Yaskawa INFORM job: OK_R2_O24A(90,180)OKKR.JBI

/JOB
//NAME OK_R2_O24A(90,180)OKKR
///FOLDERNAME X4
//POS
///NPOS 233,233,233,10,0,0
///TOOL 0
///POSTYPE PULSE
///PULSE
C00000=127652,-120361,-107124,-61599,94745,-41314
C00001=123475,-119595,-103586,-61416,91214,-41301
C00002=121798,-119103,-102107,-61373,89825,-41321
C00003=122733,-118069,-99629,-61351,89920,-40763
C00004=120759,-117967,-99269,-61347,88586,-41030
C00005=122733,-118069,-99629,-61351,89920,-40763
C00006=121798,-119103,-102107,-61373,89825,-41321
C00007=117736,-119840,-102035,-61299,87044,-41840
C00008=118269,-119289,-100643,-61321,87094,-41519
C00009=117736,-119840,-102035,-61299,87044,-41840
C00010=121798,-119103,-102107,-61373,89825,-41321
C00011=123475,-119595,-103586,-61416,91214,-41301
C00012=127652,-120361,-107124,-61599,94745,-41314
C00013=127664,-121874,-113088,-61940,96182,-42489
C00014=117115,-87413,-101371,-50413,71167,-56127
C00015=66151,-120554,-113574,30777,43812,65962
C00016=113877,-122249,-113408,59907,95932,42467
C00017=113867,-121142,-108836,59653,94764,41571
C00018=117868,-120368,-105215,59444,91320,41562
C00019=119473,-119873,-103704,59391,89968,41583
C00020=118549,-118895,-101268,59373,90014,41025
C00021=120527,-118786,-100908,59355,88700,41315
C00022=118549,-118895,-101268,59373,90014,41025
C00023=119473,-119873,-103704,59391,89968,41583
C00024=123258,-117515,-102568,59288,87895,42464
C00025=122738,-117052,-101204,59310,87899,42134
C00026=123258,-117515,-102568,59288,87895,42464
C00027=119473,-119873,-103704,59391,89968,41583
C00028=117868,-120368,-105215,59444,91320,41562
C00029=113867,-121142,-108836,59653,94764,41571
C00030=113886,-122760,-117047,60167,96954,43261
C00031=81768,-128676,-127164,-15806,118189,66385
C00032=79004,-140641,-127713,-15667,112059,66186
C00033=77808,-144944,-127724,-15696,109702,66057
C00034=77676,-143805,-125746,-15659,109067,66094
C00035=77808,-144944,-127724,-15696,109702,66057
C00036=78130,-142192,-126626,-15703,110477,66072
C00037=76506,-149132,-128502,-15827,107837,65823
C00038=78130,-142192,-126626,-15703,110477,66072
C00039=79304,-137934,-126607,-15683,112802,66198
C00040=82020,-126149,-126054,-15842,118830,66390
C00041=45668,-110490,-122952,-22349,117541,52365
C00042=41760,-118667,-122686,-21975,112477,51881
C00043=40128,-121497,-122407,-21896,110540,51637
C00044=40144,-121605,-121196,-21769,109799,51788
C00045=40128,-121497,-122407,-21896,110540,51637
C00046=39919,-122164,-122422,-21867,110176,51628
C00047=38131,-124825,-123234,-21938,108903,51193
C00048=39919,-122164,-122422,-21867,110176,51628
C00049=41560,-119373,-122718,-21939,112106,51878
C00050=45486,-111289,-123025,-22292,117155,52375
C00051=60348,-140701,-127103,-28754,99539,31549
C00052=54796,-138804,-123817,-28917,96708,30105
C00053=52592,-137758,-122419,-28964,95663,29514
C00054=52702,-137492,-121095,-28918,95104,29697
C00055=52592,-137758,-122419,-28964,95663,29514
C00056=49009,-116057,-117095,-27498,107592,27945
C00057=47407,-118890,-118021,-27463,106285,27640
C00058=49009,-116057,-117095,-27498,107592,27945
C00059=59113,-113942,-113751,-33983,108864,30548
C00060=57786,-110790,-112582,-34290,109095,29908
C00061=59113,-113942,-113751,-33983,108864,30548
C00062=61156,-113321,-114547,-33985,110341,30937
C00063=66201,-110919,-116247,-34062,114212,31827
C00064=147445,-132687,-126150,-4301,121059,-77492
C00065=147445,-132300,-123121,-4220,119399,-77426
C00066=147445,-132050,-121881,-4191,118765,-77401
C00067=147350,-132416,-123233,-4255,119403,-77464
C00068=146726,-127150,-120434,-4530,120350,-77751
C00069=147442,-131993,-121695,-3444,118967,-77377
C00070=147448,-131959,-121392,-9160,117748,-84426
C00071=147448,-132100,-122011,-9421,117974,-84714
C00072=147407,-131707,-121399,25510,108191,-66414
C00073=147408,-131563,-120771,25459,107908,-66479
C00074=147298,-131973,-122137,25545,108513,-66383
C00075=146691,-126789,-119356,25610,109561,-66381
C00076=147414,-131682,-121104,25287,108073,-66449
C00077=147414,-131822,-121732,25339,108359,-66384
C00078=147427,-132043,-122396,24992,108700,-66326
C00079=147436,-132206,-122926,23450,109836,-66194
C00080=147436,-132085,-122296,23397,109536,-66258
C00081=147412,-132364,-123624,23503,110163,-66135
C00082=146719,-127131,-120821,23546,111246,-66177
C00083=147443,-132145,-122395,23444,109538,-66252
C00084=147442,-132265,-123025,23498,109838,-66188
C00085=147459,-132404,-123153,24285,109386,-66219
C00086=147460,-132283,-122521,24231,109086,-66285
C00087=147402,-132593,-123857,24332,109710,-66171
C00088=146741,-127304,-121046,24392,110806,-66190
C00089=147467,-132359,-122683,24040,109257,-66260
C00090=147466,-132478,-123315,24094,109558,-66195
C00091=147475,-132593,-123647,23235,110203,-66122
C00092=147489,-132639,-123374,22744,111230,-65948
C00093=147489,-132524,-122773,22691,110942,-66007
C00094=147512,-132755,-124086,22814,111574,-65867
C00095=146769,-127512,-121238,22835,112649,-65938
C00096=147496,-132556,-122720,22636,111020,-65992
C00097=147495,-132672,-123318,22689,111306,-65933
C00098=147513,-132802,-123388,23030,110383,-66086
C00099=147513,-132682,-122773,22978,110090,-66147
C00100=147513,-132943,-124095,23091,110718,-66017
C00101=146792,-127670,-121267,23125,111813,-66071
C00102=147519,-132724,-122791,23106,109746,-66204
C00103=147519,-132846,-123413,23158,110041,-66143
C00104=147522,-132813,-123145,22539,111461,-65901
C00105=147523,-132659,-122379,23084,112565,-65631
C00106=147544,-133018,-123434,20123,111938,-65974
C00107=147545,-132894,-122823,20074,111643,-66027
C00108=147662,-133050,-124112,20212,112286,-65864
C00109=146819,-127879,-121296,20181,113361,-65998
C00110=147551,-132935,-122806,19750,111499,-66076
C00111=147551,-133061,-123422,19798,111796,-66023
C00112=147569,-132909,-122194,21074,111640,-65938
C00113=147569,-132763,-121591,21026,111363,-65990
C00114=147662,-133004,-122907,21158,111981,-65836
C00115=146842,-127897,-120077,21127,113017,-65960
C00116=147572,-132884,-122015,20139,111221,-66082
C00117=147578,-132996,-122335,19245,111024,-66186
C00118=147576,-133257,-123572,19337,111618,-66084
C00119=147573,-133675,-126595,19593,113174,-65811
C00120=147212,-134132,-128548,19677,114172,-65774
C00121=80085,-121932,-126319,-31537,110157,-16460
C00122=80084,-123019,-122780,-30975,107800,-15768
C00123=80084,-123205,-121288,-30786,106924,-15517
C00124=79034,-127796,-122705,-30605,105259,-15473
C00125=80112,-123119,-122506,-30931,107620,-15705
C00126=80090,-123174,-121318,-30792,106957,-15524
C00127=80091,-122983,-122809,-30981,107834,-15775
C00128=80092,-121884,-126344,-31545,110194,-16468
C00129=80173,-119669,-128927,16022,111537,-14779
C00130=80165,-121654,-125938,15693,108783,-15165
C00131=80162,-122169,-124659,15585,107769,-15304
C00132=80251,-121905,-125821,15678,108573,-15163
C00133=79115,-127188,-126213,15354,106397,-15865
C00134=80156,-122227,-124572,15576,107690,-15316
C00135=80159,-121723,-125855,15683,108701,-15179
C00136=80167,-119771,-128854,16009,111444,-14795
C00137=87390,-93317,-98199,52553,51508,-25586
C00138=80872,-118727,-107349,60414,51141,-30734
C00139=85193,-32235,-33504,-7004,70667,8141
C00140=117323,-30676,-22206,-16089,69434,20075
C00141=103961,-7641,2169,-13017,63971,15675
C00142=76008,40061,1359,-13724,89437,15522
C00143=74954,43462,7903,-13463,87051,15436
C00144=74543,44920,10634,-13367,86079,15405
C00145=73408,46552,11060,-13079,86465,14985
C00146=72826,50775,15638,-12938,85743,14869
C00147=72990,50408,15229,-12963,85836,14914
C00148=72990,49930,17364,-12980,84313,15072
C00149=74543,44920,10634,-13367,86079,15405
C00150=74691,43869,4038,-13398,89530,15082
C00151=70203,43417,5044,-20026,94803,24676
C00152=68706,45434,10156,-19691,92468,24547
C00153=68117,46334,12302,-19567,91523,24497
C00154=68118,46082,13441,-19554,90739,24624
C00155=68117,46334,12302,-19567,91523,24497
C00156=66360,47485,11887,-19269,91924,23829
C00157=65924,48399,12877,-19185,91695,23716
C00158=66360,47485,11887,-19269,91924,23829
C00159=68409,44550,4583,-19740,95210,23999
C00160=63533,47755,9354,-24595,105063,37049
C00161=61795,47183,11701,-24300,102985,36856
C00162=61100,47033,12721,-24188,102144,36779
C00163=61101,46749,13992,-24093,101295,36957
C00164=61100,47033,12721,-24188,102144,36779
C00165=59988,46978,11651,-24198,102411,36317
C00166=59669,47136,11822,-24177,102300,36224
C00167=60208,47646,12371,-24199,102381,36404
C00168=62424,47676,8250,-24625,105334,36583
C00169=81168,21826,-12659,-33512,109834,56719
C00170=78482,17537,-12923,-33053,107112,56485
C00171=78483,17226,-11558,-32863,106266,56747
C00172=78482,17537,-12923,-33053,107112,56485
C00173=77766,16655,-15276,-33240,107685,56015
C00174=77497,15571,-16273,-33245,107632,55923
C00175=77766,16655,-15276,-33240,107685,56015
C00176=80481,20983,-15004,-33739,110426,56245
C00177=67968,42334,3348,-31265,106833,14778
C00178=66287,43458,7461,-30850,104561,14772
C00179=65947,43054,8150,-30753,103897,14826
C00180=66364,43687,8867,-30739,103941,14975
C00181=65621,44273,8238,-30808,104278,14592
C00182=65959,43095,8193,-30753,103896,14831
C00183=66497,45624,10922,-29891,99696,11683
C00184=66674,44202,9408,-27708,94060,6579
C00185=67479,46599,11965,-25789,90389,3478
C00186=68273,48588,14110,-23425,86957,273
C00187=69426,50721,15271,-24933,89210,2217
C00188=70450,47061,8379,-25191,91653,2063
C00189=81534,46621,7906,-26613,118087,64927
C00190=80305,42029,5941,-26466,116681,64788
C00191=79935,40851,6052,-26330,115962,64822
C00192=80181,42155,7239,-26298,115983,64915
C00193=79800,40537,4287,-26590,116754,64562
C00194=74346,52179,18294,-26567,112715,63380
C00195=74329,52217,18336,-26567,112704,63376
C00196=73121,47301,13124,-27751,105561,55602
C00197=71250,51153,17300,-27200,100766,51701
C00198=72206,56204,21362,-27528,102760,53475
C00199=73217,55829,18030,-27817,104736,53371
C00200=73784,42190,3206,-25910,93238,2896
C00201=72676,45578,9727,-25616,90856,3024
C00202=72110,47261,12673,-25474,89830,3041
C00203=72825,45636,10952,-25632,90244,3210
C00204=72243,47296,11483,-25524,90549,2936
C00205=72123,47316,12732,-25477,89826,3046
C00206=73240,48559,14162,-23178,86629,-33
C00207=73401,47123,12578,-18501,82477,-5481
C00208=74010,47732,13368,-15080,80080,-8973
C00209=74727,48480,14235,-13386,79055,-10615
C00210=75367,48626,14271,-11603,78315,-12322
C00211=78915,50569,16259,-12822,78610,-11152
C00212=81424,51392,17049,-13667,78944,-10338
C00213=73414,33805,-5390,-8719,81797,-15206
C00214=73071,12872,-25562,-8573,83403,-15427
C00215=76462,51369,5875,-15060,108642,28273
C00216=62095,44437,5558,-29162,120992,27635
C00217=60325,42778,6723,-28941,119030,27454
C00218=61014,24421,-11522,-28546,110075,30066
C00219=60307,43049,8174,-28720,118360,27641
C00220=59612,42473,6313,-29077,118879,27193
C00221=60936,24520,-11425,-28544,110044,30045
C00222=59855,38187,2466,-28246,108344,30070
C00223=60633,45531,11034,-30883,107902,18652
C00224=60993,48477,14223,-30632,103481,15387
C00225=61232,49026,14820,-29885,99340,12011
C00226=62386,52295,16994,-30447,102054,13956
C00227=63442,52253,14034,-30764,103981,13831
C00228=65403,21797,-9707,-27343,89394,10834
C00229=66767,-521,-20868,-24959,75788,9558
C00230=89867,-61679,-55301,-17873,66984,-4382
C00231=109690,-121043,-61974,-28141,46550,4689
C00232=71363,-137537,-82431,26619,16124,-21791
BC00000=18805,363822,1075139
BC00001=18805,363822,1075139
BC00002=18805,363822,1075139
BC00003=18805,363822,1075139
BC00004=18805,363822,1075139
BC00005=18805,363822,1075139
BC00006=18805,363822,1075139
BC00007=18805,363822,1075139
BC00008=18805,363822,1075139
BC00009=18805,363822,1075139
BC00010=18805,363822,1075139
BC00011=18805,363822,1075139
BC00012=18805,363822,1075139
BC00013=18805,363822,1075139
BC00014=18805,443821,1075139
BC00015=18805,443821,1075139
BC00016=188967,363064,1075139
BC00017=188967,363064,1075139
BC00018=188967,363064,1075139
BC00019=188967,363064,1075139
BC00020=188967,363064,1075139
BC00021=188967,363064,1075139
BC00022=188967,363064,1075139
BC00023=188967,363064,1075139
BC00024=188967,363064,1075139
BC00025=188967,363064,1075139
BC00026=188967,363064,1075139
BC00027=188967,363064,1075139
BC00028=188967,363064,1075139
BC00029=188967,363064,1075139
BC00030=188967,363064,1075139
BC00031=-1,300813,1075139
BC00032=-1,300813,1075139
BC00033=-1,300813,1075139
BC00034=-1,300813,1075139
BC00035=-1,300813,1075139
BC00036=-1,300813,1075139
BC00037=-1,300813,1075139
BC00038=-1,300813,1075139
BC00039=-1,300813,1075139
BC00040=-1,300813,1075139
BC00041=57672,278687,1075139
BC00042=57672,278687,1075139
BC00043=57672,278687,1075139
BC00044=57672,278687,1075139
BC00045=57672,278687,1075139
BC00046=57672,278687,1075139
BC00047=57672,278687,1075139
BC00048=57672,278687,1075139
BC00049=57672,278687,1075139
BC00050=57672,278687,1075139
BC00051=128982,287378,1075139
BC00052=128982,287378,1075139
BC00053=128982,287378,1075139
BC00054=128982,287378,1075139
BC00055=128982,287378,1075139
BC00056=128982,287378,1075139
BC00057=128982,287378,1075139
BC00058=128982,287378,1075139
BC00059=128982,287378,1075139
BC00060=128982,287378,1075139
BC00061=128982,287378,1075139
BC00062=128982,287378,1075139
BC00063=128982,287378,1075139
BC00064=227577,310047,1075139
BC00065=229358,315236,1075139
BC00066=230071,317312,1075139
BC00067=230071,317312,1075139
BC00068=230071,317312,1075139
BC00069=232622,316461,1075139
BC00070=227204,321651,1075139
BC00071=226480,320869,1075139
BC00072=267805,316324,1075139
BC00073=267749,317413,1075139
BC00074=267749,317413,1075139
BC00075=267749,317413,1075139
BC00076=261071,317456,1075139
BC00077=261120,316369,1075139
BC00078=247856,316471,1075139
BC00079=238240,315937,1075139
BC00080=238239,317010,1075139
BC00081=238239,317010,1075139
BC00082=238239,317010,1075139
BC00083=231954,317007,1075139
BC00084=231957,315934,1075139
BC00085=214518,316147,1075139
BC00086=214479,317214,1075139
BC00087=214479,317214,1075139
BC00088=214479,317214,1075139
BC00089=207705,317131,1075139
BC00090=207735,316063,1075139
BC00091=199022,315743,1075139
BC00092=185104,314007,1075139
BC00093=185110,315129,1075139
BC00094=185110,315129,1075139
BC00095=185110,315129,1075139
BC00096=178555,314940,1075139
BC00097=178545,313814,1075139
BC00098=160848,315020,1075139
BC00099=160828,316119,1075139
BC00100=160828,316119,1075139
BC00101=160828,316119,1075139
BC00102=154951,316562,1075139
BC00103=154981,315474,1075139
BC00104=152219,313316,1075139
BC00105=151426,310632,1075139
BC00106=129622,314063,1075139
BC00107=129672,315170,1075139
BC00108=129672,315170,1075139
BC00109=129672,315170,1075139
BC00110=122930,315526,1075139
BC00111=122871,314427,1075139
BC00112=105506,312734,1075139
BC00113=105529,313869,1075139
BC00114=105529,313869,1075139
BC00115=105529,313869,1075139
BC00116=102857,314935,1075139
BC00117=96992,315999,1075139
BC00118=97677,313903,1075139
BC00119=99388,308662,1075139
BC00120=99388,308662,1075139
BC00121=25683,320032,1075139
BC00122=28530,320018,1075139
BC00123=29668,320012,1075139
BC00124=29668,320012,1075139
BC00125=29668,320012,1075139
BC00126=34209,320025,1075139
BC00127=33070,320030,1075139
BC00128=30224,320045,1075139
BC00129=85300,368981,1075139
BC00130=82937,365904,1075139
BC00131=81992,364674,1075139
BC00132=81992,364674,1075139
BC00133=81992,364674,1075139
BC00134=78116,364663,1075139
BC00135=79061,365893,1075139
BC00136=81424,368970,1075139
BC00137=81424,477665,1075139
BC00138=81424,517683,1075139
BC00139=258120,514627,389239
BC00140=273760,466775,389239
BC00141=281890,441897,389239
BC00142=268303,389739,113483
BC00143=268303,389739,113483
BC00144=268303,389739,113483
BC00145=268303,389739,113483
BC00146=268303,389739,113483
BC00147=268303,389739,113483
BC00148=268303,389739,113483
BC00149=268303,389739,113483
BC00150=268303,389739,113483
BC00151=254705,396265,114341
BC00152=254705,396265,114341
BC00153=254705,396265,114341
BC00154=254705,396264,114338
BC00155=254705,396265,114341
BC00156=254705,396265,114341
BC00157=254705,396265,114341
BC00158=254705,396265,114341
BC00159=254705,396265,114341
BC00160=229913,397396,112121
BC00161=229913,397396,112121
BC00162=229913,397396,112121
BC00163=229913,397396,112121
BC00164=229913,397396,112121
BC00165=229913,397396,112121
BC00166=229913,397396,112121
BC00167=229913,397396,112121
BC00168=229913,397396,112121
BC00169=237860,415682,113770
BC00170=237860,415682,113770
BC00171=237860,415682,113770
BC00172=237860,415682,113770
BC00173=237860,415682,113770
BC00174=237860,415682,113770
BC00175=237860,415682,113770
BC00176=237860,415682,113770
BC00177=252617,388138,87053
BC00178=252617,388138,87053
BC00179=252616,388138,87050
BC00180=252617,388138,87053
BC00181=252617,388138,87053
BC00182=252616,388138,87050
BC00183=252617,388138,87053
BC00184=252617,388138,87050
BC00185=252617,388138,87053
BC00186=252617,388138,87053
BC00187=252617,388138,87053
BC00188=252617,388138,87053
BC00189=232025,436667,94687
BC00190=232025,436667,94687
BC00191=232026,436667,94684
BC00192=232025,436667,94687
BC00193=232025,436667,94687
BC00194=232025,436667,94687
BC00195=232025,436667,94687
BC00196=232025,436667,94687
BC00197=232025,436667,94687
BC00198=232025,436667,94687
BC00199=232025,436667,94687
BC00200=264314,390036,87192
BC00201=264314,390036,87192
BC00202=264314,390035,87190
BC00203=264314,390036,87192
BC00204=264314,390036,87192
BC00205=264314,390035,87190
BC00206=264314,390036,87192
BC00207=264314,390036,87192
BC00208=264314,390036,87192
BC00209=264314,390036,87192
BC00210=264314,390036,87192
BC00211=264314,390036,87192
BC00212=264314,390036,87192
BC00213=264314,390036,87192
BC00214=264314,390036,87192
BC00215=246632,415573,91296
BC00216=234603,386738,86921
BC00217=234603,386738,86921
BC00218=234603,386738,86921
BC00219=234603,386738,86921
BC00220=234603,386738,86921
BC00221=234603,386738,86921
BC00222=234603,386738,86921
BC00223=234603,386738,86921
BC00224=234603,386738,86921
BC00225=234603,386738,86921
BC00226=234603,386738,86921
BC00227=234603,386738,86921
BC00228=240912,382948,130135
BC00229=245299,380312,160183
BC00230=270157,365379,243914
BC00231=274044,363044,357076
BC00232=274044,514823,357076
EC00000=-798156,-1296783
EC00001=-798156,-1296783
EC00002=-798156,-1296783
EC00003=-798156,-1296783
EC00004=-798156,-1296783
EC00005=-798156,-1296783
EC00006=-798156,-1296783
EC00007=-798156,-1296783
EC00008=-798156,-1296783
EC00009=-798156,-1296783
EC00010=-798156,-1296783
EC00011=-798156,-1296783
EC00012=-798156,-1296783
EC00013=-798156,-1296783
EC00014=-798156,-1296783
EC00015=-798156,-1296783
EC00016=-798156,-1296783
EC00017=-798156,-1296783
EC00018=-798156,-1296783
EC00019=-798156,-1296783
EC00020=-798156,-1296783
EC00021=-798156,-1296783
EC00022=-798156,-1296783
EC00023=-798156,-1296783
EC00024=-798156,-1296783
EC00025=-798156,-1296783
EC00026=-798156,-1296783
EC00027=-798156,-1296783
EC00028=-798156,-1296783
EC00029=-798156,-1296783
EC00030=-798156,-1296783
EC00031=-798156,-1296783
EC00032=-798156,-1296783
EC00033=-798156,-1296783
EC00034=-798156,-1296783
EC00035=-798156,-1296783
EC00036=-798156,-1296783
EC00037=-798156,-1296783
EC00038=-798156,-1296783
EC00039=-798156,-1296783
EC00040=-798156,-1296783
EC00041=-798156,-1296783
EC00042=-798156,-1296783
EC00043=-798156,-1296783
EC00044=-798156,-1296783
EC00045=-798156,-1296783
EC00046=-798156,-1296783
EC00047=-798156,-1296783
EC00048=-798156,-1296783
EC00049=-798156,-1296783
EC00050=-798156,-1296783
EC00051=-798156,-1296783
EC00052=-798156,-1296783
EC00053=-798156,-1296783
EC00054=-798156,-1296783
EC00055=-798156,-1296783
EC00056=-798156,-1296783
EC00057=-798156,-1296783
EC00058=-798156,-1296783
EC00059=-798156,-1296783
EC00060=-798156,-1296783
EC00061=-798156,-1296783
EC00062=-798156,-1296783
EC00063=-798156,-1296783
EC00064=-798156,-1296783
EC00065=-798156,-1296783
EC00066=-798156,-1296783
EC00067=-798156,-1296783
EC00068=-798156,-1296783
EC00069=-798156,-1296783
EC00070=-798156,-1296783
EC00071=-798156,-1296783
EC00072=-798156,-1296783
EC00073=-798156,-1296783
EC00074=-798156,-1296783
EC00075=-798156,-1296783
EC00076=-798156,-1296783
EC00077=-798156,-1296783
EC00078=-798156,-1296783
EC00079=-798156,-1296783
EC00080=-798156,-1296783
EC00081=-798156,-1296783
EC00082=-798156,-1296783
EC00083=-798156,-1296783
EC00084=-798156,-1296783
EC00085=-798156,-1296783
EC00086=-798156,-1296783
EC00087=-798156,-1296783
EC00088=-798156,-1296783
EC00089=-798156,-1296783
EC00090=-798156,-1296783
EC00091=-798156,-1296783
EC00092=-798156,-1296783
EC00093=-798156,-1296783
EC00094=-798156,-1296783
EC00095=-798156,-1296783
EC00096=-798156,-1296783
EC00097=-798156,-1296783
EC00098=-798156,-1296783
EC00099=-798156,-1296783
EC00100=-798156,-1296783
EC00101=-798156,-1296783
EC00102=-798156,-1296783
EC00103=-798156,-1296783
EC00104=-798156,-1296783
EC00105=-798156,-1296783
EC00106=-798156,-1296783
EC00107=-798156,-1296783
EC00108=-798156,-1296783
EC00109=-798156,-1296783
EC00110=-798156,-1296783
EC00111=-798156,-1296783
EC00112=-798156,-1296783
EC00113=-798156,-1296783
EC00114=-798156,-1296783
EC00115=-798156,-1296783
EC00116=-798156,-1296783
EC00117=-798156,-1296783
EC00118=-798156,-1296783
EC00119=-798156,-1296783
EC00120=-798156,-1296783
EC00121=-798156,-1296783
EC00122=-798156,-1296783
EC00123=-798156,-1296783
EC00124=-798156,-1296783
EC00125=-798156,-1296783
EC00126=-798156,-1296783
EC00127=-798156,-1296783
EC00128=-798156,-1296783
EC00129=-798156,-1296783
EC00130=-798156,-1296783
EC00131=-798156,-1296783
EC00132=-798156,-1296783
EC00133=-798156,-1296783
EC00134=-798156,-1296783
EC00135=-798156,-1296783
EC00136=-798156,-1296783
EC00137=-798156,-1296783
EC00138=-798156,-1296783
EC00139=-798156,-1296783
EC00140=-798156,-1296783
EC00141=-798156,-1296783
EC00142=-798156,-1296783
EC00143=-798156,-1296783
EC00144=-798156,-1296783
EC00145=-798156,-1296783
EC00146=-798156,-1296783
EC00147=-798156,-1296783
EC00148=-798156,-1296783
EC00149=-798156,-1296783
EC00150=-798156,-1296783
EC00151=-798156,-1296783
EC00152=-798156,-1296783
EC00153=-798156,-1296783
EC00154=-798154,-1296781
EC00155=-798156,-1296783
EC00156=-798156,-1296783
EC00157=-798156,-1296783
EC00158=-798156,-1296783
EC00159=-798156,-1296783
EC00160=-798156,-1296783
EC00161=-798156,-1296783
EC00162=-798156,-1296783
EC00163=-798156,-1296783
EC00164=-798156,-1296783
EC00165=-798156,-1296783
EC00166=-798156,-1296783
EC00167=-798156,-1296783
EC00168=-798156,-1296783
EC00169=-798156,-1296783
EC00170=-798156,-1296783
EC00171=-798156,-1296783
EC00172=-798156,-1296783
EC00173=-798156,-1296783
EC00174=-798156,-1296783
EC00175=-798156,-1296783
EC00176=-798156,-1296783
EC00177=-798156,-1296783
EC00178=-798156,-1296783
EC00179=-798154,-1296781
EC00180=-798156,-1296783
EC00181=-798156,-1296783
EC00182=-798154,-1296781
EC00183=-798156,-1296783
EC00184=-798155,-1296782
EC00185=-798156,-1296783
EC00186=-798156,-1296783
EC00187=-798156,-1296783
EC00188=-798156,-1296783
EC00189=-798156,-1296783
EC00190=-798156,-1296783
EC00191=-798154,-1296782
EC00192=-798156,-1296783
EC00193=-798156,-1296783
EC00194=-798156,-1296783
EC00195=-798156,-1296783
EC00196=-798156,-1296783
EC00197=-798156,-1296783
EC00198=-798156,-1296783
EC00199=-798156,-1296783
EC00200=-798156,-1296783
EC00201=-798156,-1296783
EC00202=-798155,-1296783
EC00203=-798156,-1296783
EC00204=-798156,-1296783
EC00205=-798155,-1296783
EC00206=-798156,-1296783
EC00207=-798156,-1296783
EC00208=-798156,-1296783
EC00209=-798156,-1296783
EC00210=-798156,-1296783
EC00211=-798156,-1296783
EC00212=-798156,-1296783
EC00213=-798156,-1296783
EC00214=-798156,-1296783
EC00215=-798156,-1296783
EC00216=-798156,-1296783
EC00217=-798156,-1296783
EC00218=-798156,-1296783
EC00219=-798156,-1296783
EC00220=-798156,-1296783
EC00221=-798156,-1296783
EC00222=-798156,-1296783
EC00223=-798156,-1296783
EC00224=-798156,-1296783
EC00225=-798156,-1296783
EC00226=-798156,-1296783
EC00227=-798156,-1296783
EC00228=-798156,-1296783
EC00229=-798156,-1296783
EC00230=-798156,-1296783
EC00231=-798156,-1296783
EC00232=-798156,-1296783
///POSTYPE BASE
///RECTAN
///RCONF 0,0,0,0,1,0,0,0,0,0,0,0,0,0,0,0,0,0,0,0,0,0,0,0
P00006=2.006,1.622,-0.565,0.0000,0.0000,0.0000
P00021=0.073,2.058,-0.109,0.0000,0.0000,0.0000
P00022=2.006,1.622,-0.565,0.0000,0.0000,0.0000
///RCONF 0,0,0,0,0,0,0,0,0,0,0,0,0,0,0,0,0,0,0,0,0,0,0,0
P00023=-2.957,-4.083,2.762,0.0000,0.0000,0.0000
P00024=-1.466,-0.226,-0.419,0.0000,0.0000,0.0000
P00031=-0.170,0.039,-0.647,0.0000,0.0000,0.0000
P00032=-0.423,0.157,3.222,0.0000,0.0000,0.0000
P00033=0.854,-1.099,3.047,0.0000,0.0000,0.0000
///RCONF 0,0,0,0,1,0,0,0,0,0,0,0,0,0,0,0,0,0,0,0,0,0,0,0
P00034=-8.151,9.743,-4.393,0.0000,0.0000,0.0000
///RCONF 0,0,0,0,0,0,0,0,0,0,0,0,0,0,0,0,0,0,0,0,0,0,0,0
P00035=0.390,-0.027,1.040,0.0000,0.0000,0.0000
//INST
///DATE 2024/11/18 11:58
///ATTR SC,RW
///GROUP1 RB1,BS1
///GROUP2 ST1
NOP
COMM 'OK_r2_O24A(90,180)popr
COMM 'Path S1555
COMM SFTOF3D
COMM MOVJ C00000 BC00000 VJ=100.00  +MOVJ EC00000 VJ=100.00
COMM MOVL C00001 BC00001 V=400.0  +MOVJ EC00001 VJ=100.00
COMM SMOVL C00002 BC00002 V=100.0  +MOVJ EC00002
COMM SMOVL C00003 BC00003 V=60.0  +MOVJ EC00003
COMM SREFP 3 C00004 BC00004  +REFP EC00004
COMM CALL JOB:SEARCH-R1-S13D
COMM SET P031 P006
COMM SFTON3D P031
COMM SMOVL C00005 BC00005 V=60.0  +MOVJ EC00005
COMM SMOVL C00006 BC00006 V=100.0  +MOVJ EC00006
COMM SMOVL C00007 BC00007 V=60.0  +MOVJ EC00007
COMM SREFP 3 C00008 BC00008  +REFP EC00008
COMM CALL JOB:SEARCH-R1-S13D
COMM SET P031 P006
COMM SFTON3D P031
COMM SMOVL C00009 BC00009 V=60.0  +MOVJ EC00009
COMM SMOVL C00010 BC00010 V=100.0  +MOVJ EC00010
COMM MOVL C00011 BC00011 V=400.0  +MOVJ EC00011 VJ=100.00
COMM MOVL C00012 BC00012 V=1000.0  +MOVJ EC00012 VJ=100.00
COMM MOVJ C00013 BC00013 VJ=100.00  +MOVJ EC00013 VJ=100.00
COMM MOVJ C00014 BC00014 VJ=100.00  +MOVJ EC00014 VJ=100.00
COMM MOVJ C00015 BC00015 VJ=100.00  +MOVJ EC00015 VJ=100.00
COMM MOVJ C00016 BC00016 VJ=100.00  +MOVJ EC00016 VJ=100.00
COMM 'Path S1556
COMM SFTOF3D
COMM MOVJ C00017 BC00017 VJ=100.00  +MOVJ EC00017 VJ=100.00
COMM MOVL C00018 BC00018 V=400.0  +MOVJ EC00018 VJ=100.00
COMM SMOVL C00019 BC00019 V=100.0  +MOVJ EC00019
COMM SMOVL C00020 BC00020 V=60.0  +MOVJ EC00020
COMM SREFP 3 C00021 BC00021  +REFP EC00021
COMM CALL JOB:SEARCH-R1-S13D
COMM SET P032 P006
COMM SFTON3D P032
COMM SMOVL C00022 BC00022 V=60.0  +MOVJ EC00022
COMM SMOVL C00023 BC00023 V=100.0  +MOVJ EC00023
COMM SMOVL C00024 BC00024 V=60.0  +MOVJ EC00024
COMM SREFP 3 C00025 BC00025  +REFP EC00025
COMM CALL JOB:SEARCH-R1-S13D
COMM SET P032 P006
COMM SFTON3D P032
COMM SMOVL C00026 BC00026 V=60.0  +MOVJ EC00026
COMM SMOVL C00027 BC00027 V=100.0  +MOVJ EC00027
COMM MOVL C00028 BC00028 V=400.0  +MOVJ EC00028 VJ=100.00
COMM MOVL C00029 BC00029 V=1000.0  +MOVJ EC00029 VJ=100.00
COMM MOVJ C00030 BC00030 VJ=100.00  +MOVJ EC00030 VJ=100.00
COMM 'Path S1557
COMM SFTOF3D
COMM MOVJ C00031 BC00031 VJ=100.00  +MOVJ EC00031 VJ=100.00
COMM MOVL C00032 BC00032 V=400.0  +MOVJ EC00032 VJ=100.00
COMM SMOVL C00033 BC00033 V=60.0  +MOVJ EC00033
COMM SREFP 3 C00034 BC00034  +REFP EC00034
COMM CALL JOB:SEARCH-R1-S13D
COMM SET P034 P006
COMM SFTON3D P034
COMM SMOVL C00035 BC00035 V=60.0  +MOVJ EC00035
COMM SMOVL C00036 BC00036 V=60.0  +MOVJ EC00036
COMM SREFP 3 C00037 BC00037  +REFP EC00037
COMM CALL JOB:SEARCH-R1-S13D
COMM SET P034 P006
COMM SFTON3D P034
COMM SMOVL C00038 BC00038 V=60.0  +MOVJ EC00038
COMM MOVL C00039 BC00039 V=400.0  +MOVJ EC00039 VJ=100.00
COMM MOVL C00040 BC00040 V=1000.0  +MOVJ EC00040 VJ=100.00
COMM 'Path S1558
COMM SFTOF3D
COMM MOVJ C00041 BC00041 VJ=100.00  +MOVJ EC00041 VJ=100.00
COMM MOVL C00042 BC00042 V=400.0  +MOVJ EC00042 VJ=100.00
COMM SMOVL C00043 BC00043 V=60.0  +MOVJ EC00043
COMM SREFP 3 C00044 BC00044  +REFP EC00044
COMM CALL JOB:SEARCH-R1-S13D
COMM SET P035 P006
COMM SFTON3D P035
COMM SMOVL C00045 BC00045 V=60.0  +MOVJ EC00045
COMM SMOVL C00046 BC00046 V=60.0  +MOVJ EC00046
COMM SREFP 3 C00047 BC00047  +REFP EC00047
COMM CALL JOB:SEARCH-R1-S13D
COMM SET P035 P006
COMM SFTON3D P035
COMM SMOVL C00048 BC00048 V=60.0  +MOVJ EC00048
COMM MOVL C00049 BC00049 V=400.0  +MOVJ EC00049 VJ=100.00
COMM MOVL C00050 BC00050 V=1000.0  +MOVJ EC00050 VJ=100.00
COMM 'Path S1559
COMM SFTOF3D
COMM MOVJ C00051 BC00051 VJ=100.00  +MOVJ EC00051 VJ=100.00
COMM MOVL C00052 BC00052 V=400.0  +MOVJ EC00052 VJ=100.00
COMM SMOVL C00053 BC00053 V=60.0  +MOVJ EC00053
COMM SREFP 3 C00054 BC00054  +REFP EC00054
COMM CALL JOB:SEARCH-R1-S13D
COMM SET P033 P006
COMM SFTON3D P033
COMM SMOVL C00055 BC00055 V=60.0  +MOVJ EC00055
COMM SMOVL C00056 BC00056 V=60.0  +MOVJ EC00056
COMM SREFP 3 C00057 BC00057  +REFP EC00057
COMM CALL JOB:SEARCH-R1-S13D
COMM SET P033 P006
COMM SFTON3D P033
COMM SMOVL C00058 BC00058 V=60.0  +MOVJ EC00058
COMM SMOVL C00059 BC00059 V=60.0  +MOVJ EC00059
COMM SREFP 3 C00060 BC00060  +REFP EC00060
COMM CALL JOB:SEARCH-R1-S13D
COMM SET P033 P006
COMM SFTON3D P033
COMM SMOVL C00061 BC00061 V=60.0  +MOVJ EC00061
COMM MOVL C00062 BC00062 V=400.0  +MOVJ EC00062 VJ=100.00
COMM MOVL C00063 BC00063 V=1000.0  +MOVJ EC00063 VJ=100.00
COMM 'Path W1560
COMM SFTOF3D
COMM SFTON3D P033
COMM MOVJ C00064 BC00064 VJ=100.00  +MOVJ EC00064 VJ=100.00
COMM SMOVL C00065 BC00065 V=400.0  +MOVJ EC00065
COMM SMOVL C00066 BC00066 V=100.0 PL=0  +MOVJ EC00066
COMM SREFP 1 C00067 BC00067  +REFP EC00067
COMM SREFP 2 C00068 BC00068  +REFP EC00068
COMM MACRO1 MJ#(0) ARGF0
COMM ARCON
COMM SMOVL C00069 BC00069 V=10.0  +MOVJ EC00069
COMM SMOVL C00070 BC00070 V=10.0  +MOVJ EC00070
COMM ARCOF
COMM SMOVL C00071 BC00071 V=100.0  +MOVJ EC00071
COMM SMOVL C00072 BC00072 V=100.0  +MOVJ EC00072
COMM SMOVL C00073 BC00073 V=100.0 PL=0  +MOVJ EC00073
COMM SREFP 1 C00074 BC00074  +REFP EC00074
COMM SREFP 2 C00075 BC00075  +REFP EC00075
COMM MACRO1 MJ#(0) ARGF0
COMM ARCON
COMM SMOVL C00076 BC00076 V=10.0  +MOVJ EC00076
COMM ARCOF
COMM SMOVL C00077 BC00077 V=100.0  +MOVJ EC00077
COMM SFTON3D P035
COMM SMOVL C00078 BC00078 V=100.0  +MOVJ EC00078
COMM SMOVL C00079 BC00079 V=100.0  +MOVJ EC00079
COMM SMOVL C00080 BC00080 V=100.0 PL=0  +MOVJ EC00080
COMM SREFP 1 C00081 BC00081  +REFP EC00081
COMM SREFP 2 C00082 BC00082  +REFP EC00082
COMM MACRO1 MJ#(0) ARGF0
COMM ARCON
COMM SMOVL C00083 BC00083 V=10.0  +MOVJ EC00083
COMM ARCOF
COMM SMOVL C00084 BC00084 V=100.0  +MOVJ EC00084
COMM SMOVL C00085 BC00085 V=100.0  +MOVJ EC00085
COMM SMOVL C00086 BC00086 V=100.0 PL=0  +MOVJ EC00086
COMM SREFP 1 C00087 BC00087  +REFP EC00087
COMM SREFP 2 C00088 BC00088  +REFP EC00088
COMM MACRO1 MJ#(0) ARGF0
COMM ARCON
COMM SMOVL C00089 BC00089 V=10.0  +MOVJ EC00089
COMM ARCOF
COMM SMOVL C00090 BC00090 V=100.0  +MOVJ EC00090
COMM SMOVL C00091 BC00091 V=100.0  +MOVJ EC00091
COMM SMOVL C00092 BC00092 V=100.0  +MOVJ EC00092
COMM SMOVL C00093 BC00093 V=100.0 PL=0  +MOVJ EC00093
COMM SREFP 1 C00094 BC00094  +REFP EC00094
COMM SREFP 2 C00095 BC00095  +REFP EC00095
COMM MACRO1 MJ#(0) ARGF0
COMM ARCON
COMM SMOVL C00096 BC00096 V=10.0  +MOVJ EC00096
COMM ARCOF
COMM SMOVL C00097 BC00097 V=100.0  +MOVJ EC00097
COMM SMOVL C00098 BC00098 V=100.0  +MOVJ EC00098
COMM SMOVL C00099 BC00099 V=100.0 PL=0  +MOVJ EC00099
COMM SREFP 1 C00100 BC00100  +REFP EC00100
COMM SREFP 2 C00101 BC00101  +REFP EC00101
COMM MACRO1 MJ#(0) ARGF0
COMM ARCON
COMM SMOVL C00102 BC00102 V=10.0  +MOVJ EC00102
COMM ARCOF
COMM SMOVL C00103 BC00103 V=100.0  +MOVJ EC00103
COMM SMOVL C00104 BC00104 V=100.0  +MOVJ EC00104
COMM SMOVL C00105 BC00105 V=100.0  +MOVJ EC00105
COMM SFTON3D P034
COMM SMOVL C00106 BC00106 V=100.0  +MOVJ EC00106
COMM SMOVL C00107 BC00107 V=100.0 PL=0  +MOVJ EC00107
COMM SREFP 1 C00108 BC00108  +REFP EC00108
COMM SREFP 2 C00109 BC00109  +REFP EC00109
COMM MACRO1 MJ#(0) ARGF0
COMM ARCON
COMM SMOVL C00110 BC00110 V=10.0  +MOVJ EC00110
COMM ARCOF
COMM SMOVL C00111 BC00111 V=100.0  +MOVJ EC00111
COMM SMOVL C00112 BC00112 V=100.0  +MOVJ EC00112
COMM SMOVL C00113 BC00113 V=100.0 PL=0  +MOVJ EC00113
COMM SREFP 1 C00114 BC00114  +REFP EC00114
COMM SREFP 2 C00115 BC00115  +REFP EC00115
COMM MACRO1 MJ#(0) ARGF0
COMM ARCON
COMM SMOVL C00116 BC00116 V=10.0  +MOVJ EC00116
COMM SMOVL C00117 BC00117 V=10.0  +MOVJ EC00117
COMM ARCOF
COMM SMOVL C00118 BC00118 V=400.0  +MOVJ EC00118
COMM SMOVL C00119 BC00119 V=1000.0  +MOVJ EC00119
COMM SFTOF3D
COMM MOVJ C00120 BC00120 VJ=100.00  +MOVJ EC00120 VJ=100.00
COMM 'Path W1561
COMM SFTOF3D
COMM SFTON3D P031
COMM MOVJ C00121 BC00121 VJ=100.00  +MOVJ EC00121 VJ=100.00
COMM SMOVL C00122 BC00122 V=400.0  +MOVJ EC00122
COMM SMOVL C00123 BC00123 V=100.0 PL=0  +MOVJ EC00123
COMM SREFP 1 C00124 BC00124  +REFP EC00124
COMM SREFP 2 C00125 BC00125  +REFP EC00125
COMM MACRO1 MJ#(0) ARGF0
COMM ARCON
COMM SMOVL C00126 BC00126 V=10.0  +MOVJ EC00126
COMM ARCOF
COMM SMOVL C00127 BC00127 V=400.0  +MOVJ EC00127
COMM SMOVL C00128 BC00128 V=1000.0  +MOVJ EC00128
COMM SFTOF3D
COMM 'Path W1562
COMM SFTOF3D
COMM SFTON3D P032
COMM MOVJ C00129 BC00129 VJ=100.00  +MOVJ EC00129 VJ=100.00
COMM SMOVL C00130 BC00130 V=400.0  +MOVJ EC00130
COMM SMOVL C00131 BC00131 V=100.0 PL=0  +MOVJ EC00131
COMM SREFP 1 C00132 BC00132  +REFP EC00132
COMM SREFP 2 C00133 BC00133  +REFP EC00133
COMM MACRO1 MJ#(0) ARGF0
COMM ARCON
COMM SMOVL C00134 BC00134 V=10.0  +MOVJ EC00134
COMM ARCOF
COMM SMOVL C00135 BC00135 V=400.0  +MOVJ EC00135
COMM SMOVL C00136 BC00136 V=1000.0  +MOVJ EC00136
COMM SFTOF3D
COMM MOVJ C00137 BC00137 VJ=100.00  +MOVJ EC00137 VJ=100.00
COMM MOVJ C00138 BC00138 VJ=100.00  +MOVJ EC00138 VJ=100.00
MOVJ C00139 BC00139 VJ=100.00  +MOVJ EC00139 VJ=100.00
MOVJ C00140 BC00140 VJ=100.00  +MOVJ EC00140 VJ=25.00
MOVJ C00141 BC00141 VJ=100.00  +MOVJ EC00141 VJ=100.00
SSFTOF
SFTOF
'Path S1563
SFTOF3D
MOVJ C00142 BC00142 VJ=100.00  +MOVJ EC00142 VJ=100.00
MOVL C00143 BC00143 V=666.7  +MOVJ EC00143 VJ=100.00
SMOVL C00144 BC00144 V=166.7  +MOVJ EC00144
SMOVL C00145 BC00145 V=166.7  +MOVJ EC00145
SREFP 3 C00146 BC00146  +REFP EC00146
CALL JOB:SEARCH-R1-S13D
SET P021 P006
SFTON3D P021
SMOVL C00147 BC00147 V=166.7  +MOVJ EC00147
SREFP 3 C00148 BC00148  +REFP EC00148
CALL JOB:SEARCH-R1-S13D
SET P021 P006
SFTON3D P021
SMOVL C00149 BC00149 V=166.7  +MOVJ EC00149
MOVL C00150 BC00150 V=1000.0  +MOVJ EC00150 VJ=100.00
'Path S1564
SFTOF3D
MOVJ C00151 BC00151 VJ=100.00  +MOVJ EC00151 VJ=100.00
MOVL C00152 BC00152 V=400.0  +MOVJ EC00152 VJ=100.00
SMOVL C00153 BC00153 V=166.7  +MOVJ EC00153
SREFP 3 C00154 BC00154  +REFP EC00154
CALL JOB:SEARCH-R1-S13D
SET P022 P006
SFTON3D P022
SMOVL C00155 BC00155 V=166.7  +MOVJ EC00155
SMOVL C00156 BC00156 V=166.7  +MOVJ EC00156
SREFP 3 C00157 BC00157  +REFP EC00157
CALL JOB:SEARCH-R1-S13D
SET P022 P006
SFTON3D P022
SMOVL C00158 BC00158 V=166.7  +MOVJ EC00158
MOVL C00159 BC00159 V=1000.0  +MOVJ EC00159 VJ=100.00
'Path S1565
SFTOF3D
MOVJ C00160 BC00160 VJ=100.00  +MOVJ EC00160 VJ=100.00
MOVL C00161 BC00161 V=666.7  +MOVJ EC00161 VJ=100.00
SMOVL C00162 BC00162 V=166.7  +MOVJ EC00162
SREFP 3 C00163 BC00163  +REFP EC00163
CALL JOB:SEARCH-R1-S13D
SET P023 P006
SFTON3D P023
SMOVL C00164 BC00164 V=166.7  +MOVJ EC00164
SMOVL C00165 BC00165 V=166.7  +MOVJ EC00165
SREFP 3 C00166 BC00166  +REFP EC00166
CALL JOB:SEARCH-R1-S13D
SET P023 P006
SFTON3D P023
SMOVL C00167 BC00167 V=166.7  +MOVJ EC00167
MOVL C00168 BC00168 V=1000.0  +MOVJ EC00168 VJ=100.00
'Path S1573
SFTOF3D
MOVJ C00169 BC00169 VJ=100.00  +MOVJ EC00169 VJ=100.00
SMOVL C00170 BC00170 V=166.7  +MOVJ EC00170
SREFP 3 C00171 BC00171  +REFP EC00171
CALL JOB:SEARCH-R1-S13D
SET P024 P006
SFTON3D P024
SMOVL C00172 BC00172 V=166.7  +MOVJ EC00172
SMOVL C00173 BC00173 V=166.7  +MOVJ EC00173
SREFP 3 C00174 BC00174  +REFP EC00174
CALL JOB:SEARCH-R1-S13D
SET P024 P006
SFTON3D P024
SMOVL C00175 BC00175 V=166.7  +MOVJ EC00175
MOVL C00176 BC00176 V=1000.0  +MOVJ EC00176 VJ=100.00
'Path W1571
SFTOF3D
SFTON3D P022
MOVJ C00177 BC00177 VJ=100.00  +MOVJ EC00177 VJ=100.00
SMOVL C00178 BC00178 V=666.7  +MOVJ EC00178
SMOVL C00179 BC00179 V=166.7 PL=0  +MOVJ EC00179
SREFP 1 C00180 BC00180  +REFP EC00180
SREFP 2 C00181 BC00181  +REFP EC00181
MACRO1 MJ#(0) ARGF21
ARCON
SWVON WEV#(100)
SMOVC C00182 BC00182 V=9.2  +MOVJ EC00182
SMOVC C00183 BC00183 V=8.3  +MOVJ EC00183
SMOVC C00184 BC00184 V=8.3  +MOVJ EC00184
SMOVC C00185 BC00185 V=8.3  +MOVJ EC00185
SMOVC C00186 BC00186 V=8.3  +MOVJ EC00186
ARCOF
SWVOF
SMOVL C00187 BC00187 V=400.0  +MOVJ EC00187
SMOVL C00188 BC00188 V=1000.0  +MOVJ EC00188
SFTOF3D
SFTON3D P024
MOVJ C00189 BC00189 VJ=100.00  +MOVJ EC00189 VJ=100.00
SMOVL C00190 BC00190 V=666.7  +MOVJ EC00190
SMOVL C00191 BC00191 V=166.7 PL=0  +MOVJ EC00191
SREFP 1 C00192 BC00192  +REFP EC00192
SREFP 2 C00193 BC00193  +REFP EC00193
MACRO1 MJ#(0) ARGF21
ARCON
SWVON WEV#(100)
SMOVL C00194 BC00194 V=8.3  +MOVJ EC00194
SMOVC C00195 BC00195 V=8.3  +MOVJ EC00195
SMOVC C00196 BC00196 V=8.3  +MOVJ EC00196
SMOVC C00197 BC00197 V=8.3  +MOVJ EC00197
ARCOF
SWVOF
SMOVL C00198 BC00198 V=400.0  +MOVJ EC00198
SMOVL C00199 BC00199 V=1000.0  +MOVJ EC00199
SFTOF3D
'Path W1572
SFTOF3D
SFTON3D P021
MOVJ C00200 BC00200 VJ=100.00  +MOVJ EC00200 VJ=100.00
SMOVL C00201 BC00201 V=666.7  +MOVJ EC00201
SMOVL C00202 BC00202 V=166.7 PL=0  +MOVJ EC00202
SREFP 1 C00203 BC00203  +REFP EC00203
SREFP 2 C00204 BC00204  +REFP EC00204
ARCON
SWVON WEV#(100)
SMOVC C00205 BC00205 V=8.3  +MOVJ EC00205
SMOVC C00206 BC00206 V=9.2  +MOVJ EC00206
SMOVC C00207 BC00207 V=8.3  +MOVJ EC00207
SMOVC C00208 BC00208 V=8.3  +MOVJ EC00208
SMOVC C00209 BC00209 V=8.3  +MOVJ EC00209
SMOVC C00210 BC00210 V=8.3  +MOVJ EC00210
SMOVC C00211 BC00211 V=8.3  +MOVJ EC00211
SMOVC C00212 BC00212 V=8.3  +MOVJ EC00212
ARCOF
SWVOF
SFTOF3D
SMOVL C00213 BC00213 V=400.0  +MOVJ EC00213
SMOVL C00214 BC00214 V=1000.0  +MOVJ EC00214
MOVJ C00215 BC00215 VJ=100.00  +MOVJ EC00215 VJ=100.00
SFTOF3D
SFTON3D P023
MOVJ C00216 BC00216 VJ=100.00  +MOVJ EC00216 VJ=100.00
SMOVL C00217 BC00217 V=666.7  +MOVJ EC00217
SMOVL C00218 BC00218 V=166.7 PL=0  +MOVJ EC00218
SREFP 1 C00219 BC00219  +REFP EC00219
SREFP 2 C00220 BC00220  +REFP EC00220
MACRO1 MJ#(0) ARGF21
ARCON
SWVON WEV#(100)
SMOVC C00221 BC00221 V=9.2  +MOVJ EC00221
SMOVC C00222 BC00222 V=9.2  +MOVJ EC00222
SMOVC C00223 BC00223 V=9.2  +MOVJ EC00223
SMOVC C00224 BC00224 V=9.2  +MOVJ EC00224
SMOVC C00225 BC00225 V=9.2  +MOVJ EC00225
ARCOF
SWVOF
SMOVL C00226 BC00226 V=400.0  +MOVJ EC00226
SMOVL C00227 BC00227 V=1000.0  +MOVJ EC00227
SFTOF3D
MOVJ C00228 BC00228 VJ=100.00  +MOVJ EC00228 VJ=100.00
MOVJ C00229 BC00229 VJ=100.00  +MOVJ EC00229 VJ=100.00
MOVJ C00230 BC00230 VJ=100.00  +MOVJ EC00230 VJ=100.00
MOVJ C00231 BC00231 VJ=100.00  +MOVJ EC00231 VJ=100.00
MOVJ C00232 BC00232 VJ=100.00  +MOVJ EC00232 VJ=100.00
END
